INTERFACE ITF_Control1_HMI_Connector EXTENDS 
	ITF_BaseControlElement_HMI_Connector, ITF_Control1_HMI_Connector_View, ITF_Control1_HMI_Connector_Command

END_INTERFACE

(* stored: Version 1.1.0.1
   Itf ITF_Control1_HMI_Connector: Id {b09e6ae4-cba7-048b-302b-f8d71c0e958d} *)
